# EPICS autosave request: ADApp/Db/NDStdArrays_settings.req
$(P)$(R)ArrayData.TSE
